Staubli VAL3: start.pgx

program start()
  local num l_nCounter
  local bool l_bLatched
  local string l_sMessage
begin
  cls()
  userPage()
  call create(0,"encoder")
  do
    call getValue(false,l_nCounter)
    l_sMessage="Instant val: "+toString("10",l_nCounter)
    gotoxy(5,0)
    putln(l_sMessage)
    call isLatched(l_bLatched)
    if l_bLatched==true
      call getValue(true,l_nCounter)
      l_sMessage="Latched val: "+toString("10",l_nCounter)
      gotoxy(5,1)
      putln(l_sMessage)
    endIf
    //
    l_sMessage="IsLatched: "
    if diEncLatched==true
      l_sMessage=l_sMessage+"TRUE"
    else
      l_sMessage=l_sMessage+"FALSE"
    endIf
    gotoxy(5,2)
    putln(l_sMessage)
    delay(0)
  until false
end
